PROGRAM prgMAIN
VAR
	(* Sonstiges *)
	fbZeitstempel	:	FB_Zeitstempel;
END_VAR


	fbZeitstempel();

END_PROGRAM

(* stored: Version 1.1.0.1, ProductVersion 3.1.4024.12
   POU prgMAIN: Id {e6d00dc8-42d8-40ed-9265-2c8ae6cce6a1}, SpecialFunc None *)
